FUNCTION_BLOCK FT_PID_STERI
VAR_INPUT
	T_ERR_C	: REAL;					//Error
	// Cell
	K_P_C 	: REAL := 1.0;		
	K_I_C 	: REAL := 1.0;
	K_D_C 	: REAL := 1.0;
	T_R_C	: REAL := 1.0; 			//Tracking time used for Anti-Wind up
	LIM_L 	: REAL := 0.0;			//Min. PWM
	LIM_H 	: REAL := 1.0;			//Max. PWM
	RST 	: BOOL;
END_VAR
VAR_OUTPUT
	Y 		: REAL;
	LIM 	: BOOL;
END_VAR
VAR
	//For Cell
	P_C 	: REAL;			//Proportional term
	I_C 	: REAL;			//Integral term
	D_C 	: REAL;			//Derivate term
	err_sum : REAL :=0;		//error for I
	err_k_1 : REAL :=0;		//old error
	
	
	//Saturation
	y_k		: REAL;			//control signal 
	y_sat   : REAL;			//Control signal after saturation
	y_k_1 	: REAL;			//Control signal (k-1)
	y_sat_k_1 :REAL;		//control signal after saturation (k-1)
	
	I_C_k_1	: REAL ; 		//I-Part old
	
	tx		: DWORD;
	T_a		: REAL;			//Sampling Time
	t_last	: DWORD;
END_VAR

(* if rst then *)
IF rst THEN		//Reset -- tbd
	err_sum:=0;
	err_k_1:=0;
	t_last := T_PLC_US();
	T_a := 0.0;
ELSE
	//read last cycle time in Microseconds
	tx := T_PLC_US();
	T_a := DWORD_TO_REAL(tx - t_last);
	t_last := tx;
	
	//proportional term
	P_C := K_P_C*T_ERR_C;
	
	//Integrator term with Anti-Windup backcalculation
	err_sum:=err_k_1+T_ERR_C;
	I_C := I_C_k_1 + K_I_C * err_sum * T_a/2.0 + (T_a/T_R_C)*(y_k-y_sat+y_k_1-y_sat_k_1);
	
	//Derivative term
	D_C := K_D_C * (T_ERR_C-err_k_1)/T_a;
	
	//output before saturation
	y_k := P_C + I_C + D_C;
	
	//Saturation used to limit Jacket temp.
	IF LIM_H < y_k THEN
		y_sat:= LIM_H;
	ELSIF  LIM_L > y_k THEN
		y_sat:= LIM_L;
	ELSE
		y_sat:= y_k;
	END_IF	
	
	//setting output
	Y	:= y_sat;	
	
	//save variable for next step
	I_C_k_1 := I_C;				//Saving Integral part for next step
	err_k_1 := T_ERR_C;			//Saving error for ...
END_IF

END_FUNCTION_BLOCK

(* stored: Version 1.1.0.1, ProductVersion 3.1.4022.12
   POU FT_PID_STERI: Id {8255bb89-d6ff-4fbe-925c-11e68dcf57de}, SpecialFunc None *)
